FUNCTION_BLOCK CROSSCOMM_PEER_195F5B05D36C14041 (* Service Interface Function Block Type *)
  (* Standard: 61499-2 *)
  (* Version 0.0, 9/22/2017, bababen, nxtControl GmbH, template *)
  PACKAGE Main;
  (* Compiler Cpp nxtControl builtin 1.0 *)
  {SET_ATTRIBUTE(Runtime.FBType.ImplementingType, Runtime.System#DYNGEN_CROSSCOMM_PEER)}
  {SET_ATTRIBUTE(Configuration.GenericFBType.InterfaceParams, Runtime.System#<InterfaceList> <EventOutputs> <Event Name="CNF"> <With Var="PusherRetractedCNF" /> <With Var="PusherExtendedCNF" /> </Event> </EventOutputs> <OutputVars> <VarDeclaration Name="PusherRetractedCNF" Type="BOOL" /> <VarDeclaration Name="PusherExtendedCNF" Type="BOOL" /> </OutputVars> </InterfaceList>)}
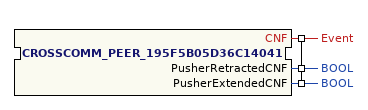
  EVENT_OUTPUT
    CNF WITH PusherRetractedCNF, PusherExtendedCNF;
  END_EVENT
  VAR_OUTPUT
    PusherRetractedCNF : BOOL;
    PusherExtendedCNF : BOOL;
  END_VAR
  EC_STATES
    START;
  END_STATES
END_FUNCTION_BLOCK
